{attribute 'strict'}
TYPE E_FixtureStateInit :
(
	FIXTURE_INIT_CLAMP	:= 0,	(*  *)
	FIXTURE_INIT_COVER	:= 20,	(*  *)
	FIXTURE_INIT_DONE	:= 10	(*  *)
);
END_TYPE

(* stored: Version 1.1.0.1, ProductVersion 3.1.4024.9
   DUT E_FixtureStateInit: Id {f09a7a78-c45e-4592-a781-c54baf08d516} *)
